FUNCTION_BLOCK Pato IMPLEMENTS I_AveVoladora, I_AveNadadora
VAR_INPUT
    velocidad : REAL;
    alturaMaxima : REAL;
    tiempoBuceo : TIME;
END_VAR
VAR
END_VAR


METHOD Nadar : BOOL
Nadar := TRUE;
END_METHOD


METHOD Volar : BOOL
Volar := true;
END_METHOD

END_FUNCTION_BLOCK

(* stored: Version 1.1.0.1, ProductVersion 3.1.4024.12
   POU Pato: Id {53750461-4c20-4932-892c-560a881fa5db}, SpecialFunc None
   Method Nadar: Id {3eb04696-5ac5-4f2e-a2e8-2f94fa5b5f7d}
   Method Volar: Id {4d4e674f-b9bd-4df3-9340-a8aeee463f30} *)
